{attribute 'qualified_only'}
VAR_GLOBAL
		//Axis: AXIS_REF;
END_VAR

(* stored: Version 1.1.0.1, ProductVersion 3.1.4024.0
   GVL gHW: Id {20abb9f4-0217-4e7d-9a2f-1ceca04bc222} *)
